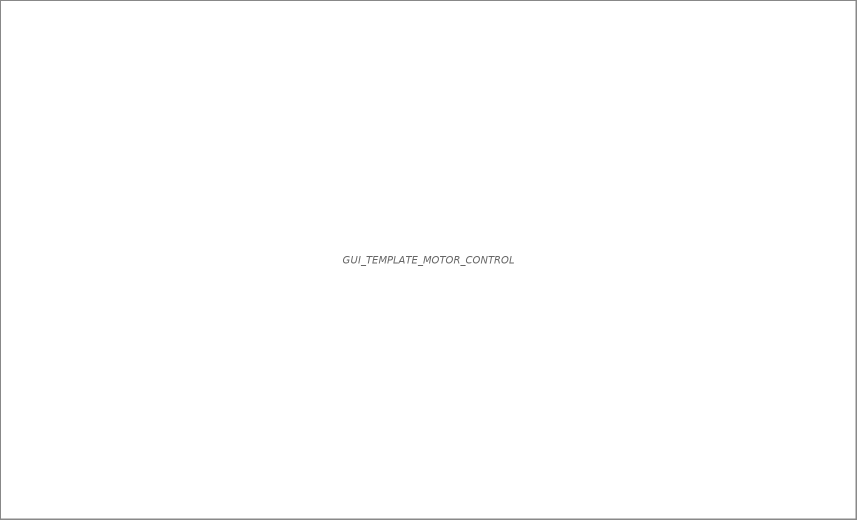
VISUALIZATION GUI_ADC_Motor1  // 857x520
    Frame (0,0 857x520)
        shows GUI_TEMPLATE_MOTOR_CONTROL(m_Instance := MAIN.adc.motor1)
END_VISUALIZATION

(* stored: Version 1.1.0.1, ProductVersion 3.1.4024.3
   Visu GUI_ADC_Motor1: Id {07e8ed33-a2aa-42f4-87e8-7760e3f8a85a} *)
